{attribute 'GeneratedUsingTerminal: EL5021-0000-0016'}
{attribute addProperty BoxType "EL5021-0000-0016"}
{attribute addProperty Id "ControlAT %Q*Control_D500AB792Set_counter_valueAT %Q*UDINT4"}
{attribute addProperty CRC "1692227694"}
{attribute addProperty Size "6"}
TYPE ENC_Control_64DD586E :
STRUCT
	{attribute addProperty Name "Control"}
	Control AT %Q* : Control_D500AB79;
	{attribute addProperty Name "Set_counter_value"}
	Set_counter_value AT %Q* : UDINT;
END_STRUCT
END_TYPE

(* stored: Version 1.2.0.0, ProductVersion 3.1.4024.9
   DUT ENC_Control_64DD586E: Id {4f1e979a-5548-4d45-b0ef-d2e20a9de50b} *)
